{attribute addProperty BoxType "AMP8000-0000-0103-0103"}
{attribute addProperty Id "Ch_A_Target_positionAT %Q*DINT3240Ch_A_Target_velocityAT %Q*DINT3240"}
{attribute addProperty CRC "1886493079"}
{attribute addProperty SizeInBites "64"}
{attribute addProperty SizeInBytes "8"}
TYPE Ch_A_Interpolator_Outputs_70719997 :
STRUCT
	{attribute addProperty Name "Ch_A_Target_position"}
	Ch_A_Target_position AT %Q* : DINT;
	{attribute addProperty Name "Ch_A_Target_velocity"}
	Ch_A_Target_velocity AT %Q* : DINT;
END_STRUCT
END_TYPE

(* stored: Version 1.2.0.0, ProductVersion 3.1.4024.9
   DUT Ch_A_Interpolator_Outputs_70719997: Id {d4a9145e-4569-49ba-aaf4-117ec0ea42bb} *)
